Staubli VAL3: robot2PC.pgx

program robot2PC()
begin

  clearBuffer(sktoPC)
  sktoPC="run"
  sDataPC=sktoPC
  _bVisionOK=true
end
